(* Logix 5000 project; controller Machine_Maintenance_Lab2 vendor 1 type 14 code 155 rev 36.11; software revision 36.00 *)

TASK MainTask (continuous, watchdog 500 ms) : MainProgram

MODULES
   Local : vendor 1 type 14 code 155 (PointIO 0, rev 36.11)
      Discrete_IO : Embedded (PointIO 1, rev 36.11, Output RPI 20 ms)
END_MODULES

PROGRAM MainProgram   (* main routine MainRoutine *)
VAR
   counter : COUNTER := (PRE := 5);
   CycleCounter : COUNTER := (PRE := 5);
   delay : TIMER := (PRE := 10);
   HighCycleTimer : COUNTER := (PRE := 700);
   i_CycleDone : ALIAS FOR o_CycleDone;
   i_GreenPB : ALIAS FOR Local:1:I.Data.0;
   i_GreenPB_ConveyorStart : ALIAS FOR i_GreenPB;
   i_GreenPBLight_Conveyor1ON : ALIAS FOR o_GreenPBLight_Conveyor1ON;
   i_Pause : ALIAS FOR Pause;
   i_Piston : ALIAS FOR Local:1:O.Data.2;
   i_RedPB_StopButton : ALIAS FOR Local:1:I.Data.1;
   i_RedPBLight_Conveyor2ON : ALIAS FOR o_RedPBLight_Conveyor2ON;
   i_Turnkey : ALIAS FOR Local:1:I.Data.2;
   i_Turnkey_ItemSensor : ALIAS FOR i_Turnkey;
   ItemCounter1 : COUNTER := (PRE := 5);
   ItemCounterLeft : COUNTER := (PRE := 5);
   ItemCounterRight : COUNTER := (PRE := 6);
   LowCycleTimer : COUNTER := (PRE := 300);
   NewCycle : BOOL;
   o_CycleDone : BOOL;
   o_GreenPBLight : ALIAS FOR Local:1:O.Data.0;
   o_GreenPBLight_Conveyor1ON : ALIAS FOR o_GreenPBLight;
   o_Piston : ALIAS FOR i_Piston;
   o_RedPBLight : ALIAS FOR Local:1:O.Data.1;
   o_RedPBLight_Conveyor2ON : ALIAS FOR o_RedPBLight;
   OS_Out : BOOL;
   Pause : BOOL;
   ResetDelay : TIMER := (PRE := 500);
   ThreeSecTimer : TIMER := (PRE := 3000);
   timer : TIMER := (PRE := 5000);
   TimerHighCycle : TIMER := (PRE := 700);
   TimerLowCycle : TIMER := (PRE := 300);
   TurnkeyOneShot : BOOL;
END_VAR

ROUTINE MainRoutine   (* ladder *)
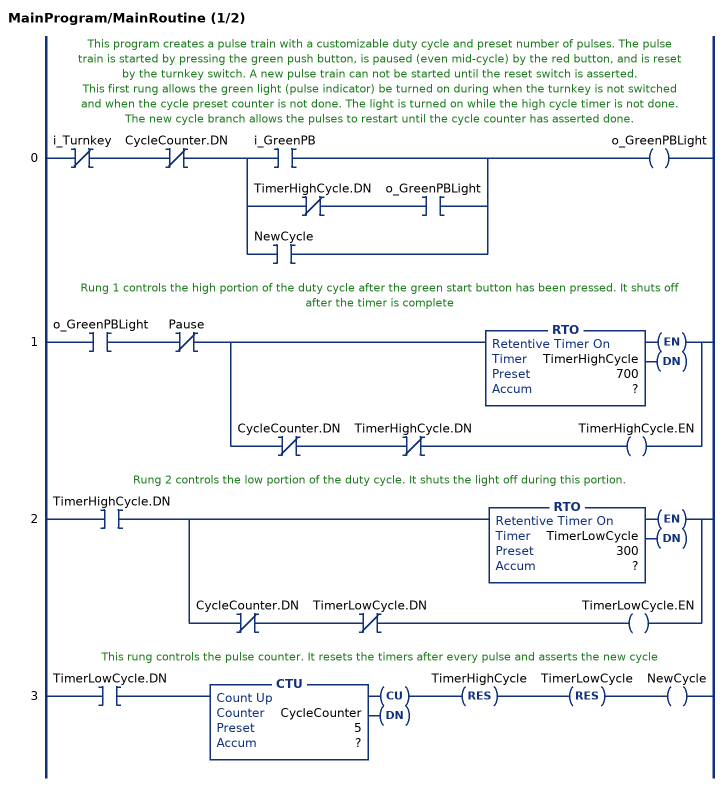
   // This program creates a pulse train with a customizable duty cycle and preset number of pulses. The pulse train is started by pressing the green push button, is paused (even mid-cycle) by the red button, and is reset by the turnkey switch. A new pulse train can not be started until the reset switch is asserted.
   // This first rung allows the green light (pulse indicator) be turned on during when the turnkey is not switched and when the cycle preset counter is not done. The light is turned on while the high cycle timer is not done. The new cycle branch allows the pulses to restart until the cycle counter has asserted done.
   0: XIO(i_Turnkey)XIO(CycleCounter.DN)[XIC(i_GreenPB) ,[XIO(TimerHighCycle.DN) XIC(o_GreenPBLight) ,XIC(NewCycle) ] ]OTE(o_GreenPBLight);
   // Rung 1 controls the high portion of the duty cycle after the green start button has been pressed. It shuts off after the timer is complete
   1: XIC(o_GreenPBLight)XIO(Pause)[RTO(TimerHighCycle,?,?) ,XIO(CycleCounter.DN) XIO(TimerHighCycle.DN) OTE(TimerHighCycle.EN) ];
   // Rung 2 controls the low portion of the duty cycle. It shuts the light off during this portion.
   2: XIC(TimerHighCycle.DN)[RTO(TimerLowCycle,?,?) ,XIO(CycleCounter.DN) XIO(TimerLowCycle.DN) OTE(TimerLowCycle.EN) ];
   // This rung controls the pulse counter. It resets the timers after every pulse and asserts the new cycle
   3: XIC(TimerLowCycle.DN)CTU(CycleCounter,?,?)RES(TimerHighCycle)RES(TimerLowCycle)OTE(NewCycle);
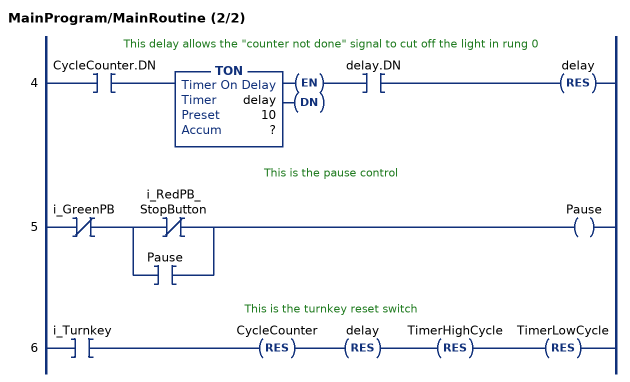
   // This delay allows the "counter not done" signal to cut off the light in rung 0
   4: XIC(CycleCounter.DN)TON(delay,?,?)XIC(delay.DN)RES(delay);
   // This is the pause control
   5: XIO(i_GreenPB)[XIO(i_RedPB_StopButton) ,XIC(Pause) ]OTE(Pause);
   // This is the turnkey reset switch
   6: XIC(i_Turnkey)RES(CycleCounter)RES(delay)RES(TimerHighCycle)RES(TimerLowCycle);
END_ROUTINE
END_PROGRAM
